FUNCTION_BLOCK RFC_TransferWorkpieceTo_PSEnd EXTENDS RFC_MoveWorkpiece_Base
VAR_INPUT
END_VAR
VAR_OUTPUT
END_VAR
VAR
	// EProcessVariables.SSC_WPAtEnd = TRUE
	m_precondition: ComparisonExpression(EProcessVariables.SSC_WPAtEnd, EComparisonType.equals, EDataType.binary, TRUE, 0, '', TRUE);
	
	// EProcessVariables.RFC_WPAtEnd = TRUE
	m_postcondition: ComparisonExpression(EProcessVariables.RFC_WPAtEnd, EComparisonType.equals, EDataType.binary, TRUE, 0, '', TRUE);
END_VAR

SUPER^();

METHOD PROTECTED  AtTarget : BOOL
VAR_INPUT
END_VAR
AtTarget := FALSE;
IF m_ptrRFC^.WPAtEnd THEN
	AtTarget := TRUE;
END_IF
END_METHOD

METHOD FB_init : BOOL
VAR_INPUT
	bInitRetains : BOOL; // if TRUE, the retain variables are initialized (warm start / cold start)
	bInCopyCode : BOOL;  // if TRUE, the instance afterwards gets moved into the copy code (online change)
	
	i_ptrRFC: POINTER TO RefeedingConveyor;
END_VAR
m_ptrRFC := i_ptrRFC;

m_id := EPrimitives.RFC_TransferWorkpieceTo_PSEnd;
m_timeout := T#200S;

Precondition := m_precondition;
Postcondition := m_postcondition;
END_METHOD

END_FUNCTION_BLOCK

(* stored: Version 1.1.0.1
   POU RFC_TransferWorkpieceTo_PSEnd: Id {49f1be7f-cf24-4eb0-8294-4bfd96bf8e22}, SpecialFunc None
   Method AtTarget: Id {75a834cf-6eb0-4855-806a-1dc8739b44df}
   Method FB_init: Id {f9c83286-1e1b-485e-bb40-08316362c9bf} *)
